{attribute 'qualified_only'}
{attribute 'strict'}
TYPE eP_ejevacMode :
(
	vacON := 1,
	vacOff := 2,
	break := 3,
	breakOff := 4,
	halt := 0
);
END_TYPE

(* stored: Version 1.1.0.1, ProductVersion 3.1.4024.11
   DUT eP_ejevacMode: Id {f5be6ee2-ab5f-4d6e-a529-13afd437d332} *)
